// TIA Portal V20 export
DATA_BLOCK "Side_Shifters_SS1"   // DB26
// stored: InstanceOfName Side_Shifters, InstanceOfType FB
"Side_Shifters"
   // VAR_INPUT
   //    set_Hydraulic_Up { ExternalAccessible := 'False'; ExternalVisible := 'False'; ExternalWritable := 'False'} : Bool;
   //    set_Hydraulic_Down { ExternalAccessible := 'False'; ExternalVisible := 'False'; ExternalWritable := 'False'} : Bool;
   //    set_SL_Hydraulic_Up : Bool;
   //    set_SL_Hydraulic_Down : Bool;
   //    set_SR_Hydraulic_Up : Bool;
   //    set_SR_Hydraulic_Down : Bool;
   //    set_SL_Hydraulic_Unit : Bool;
   //    set_SR_Hydraulic_Unit : Bool;
   //    set_Go_To_ST1 : Bool;
   //    set_Go_To_ST2 : Bool;
   //    set_Go_To_ST3 : Bool;
   //    set_Go_To_ST4 : Bool;
   //    ST1_Empty : Bool;
   //    ST2_Empty : Bool;
   //    ST3_Empty : Bool;
   //    ST4_Empty : Bool;
   //    Homing_1_SR : Int;
   //    Homing_2_SR : Int;
   //    Homing_3_SR : Int;
   //    Homing_4_SR : Int;
   //    Homing_1_SL : Int;
   //    Homing_2_SL : Int;
   //    Homing_3_SL : Int;
   //    Homing_4_SL : Int;
   //    SL_Drive_Forward : Bool;
   //    SL_Drive_Backward : Bool;
   //    SR_Drive_Forward : Bool;
   //    SR_Drive_Backward : Bool;
   //    iSL_Sen_Drv_1 : Bool;
   //    iSL_Sen_Drv_2 : Bool;
   //    iSL_Sen_Drv_3 : Bool;
   //    iSL_Sen_Drv_4 : Bool;
   //    iSR_Sen_Drv_1 : Bool;
   //    iSR_Sen_Drv_2 : Bool;
   //    iSR_Sen_Drv_3 : Bool;
   //    iSR_Sen_Drv_4 : Bool;
   //    iSL_Sen_Val1_Up : Bool;
   //    iSL_Sen_Val1_Down : Bool;
   //    iSL_Sen_Val2_Up : Bool;
   //    iSL_Sen_Val2_Down : Bool;
   //    iSR_Sen_Val1_Up : Bool;
   //    iSR_Sen_Val1_Down : Bool;
   //    iSR_Sen_Val2_Up : Bool;
   //    iSR_Sen_Val2_Down : Bool;
   //    iSL_Distance : Int;
   //    iSR_Correct : Int;
   //    iSR_Distance : Int;
   //    iSL_Hydraulic_Filtr : Bool;
   //    iSR_Hydraulic_Empty : Bool;
   //    HWIdentSL : HW_IO;
   //    HWIdentSR : HW_IO;
   //    Reset_Drive : Bool;
   //    Reset_Hydro : Bool;
   // END_VAR
   // VAR_OUTPUT
   //    oSL_Valve_Up { ExternalAccessible := 'False'; ExternalVisible := 'False'; ExternalWritable := 'False'} : Bool;
   //    oSL_Valve_Down { ExternalAccessible := 'False'; ExternalVisible := 'False'; ExternalWritable := 'False'} : Bool;
   //    oSL_Hydraulic_Unit { ExternalAccessible := 'False'; ExternalVisible := 'False'; ExternalWritable := 'False'} : Bool;
   //    oSR_Valve_Up { ExternalAccessible := 'False'; ExternalVisible := 'False'; ExternalWritable := 'False'} : Bool;
   //    oSR_Valve_Down { ExternalAccessible := 'False'; ExternalVisible := 'False'; ExternalWritable := 'False'} : Bool;
   //    oSR_Hydraulic_Unit { ExternalAccessible := 'False'; ExternalVisible := 'False'; ExternalWritable := 'False'} : Bool;
   //    oHydraulic_Status_LED_UP_1 : Bool;
   //    oHydraulic_Status_LED_UP_2 : Bool;
   //    oHydraulic_Status_LED_DOWN_1 : Bool;
   //    oHydraulic_Status_LED_DOWN_2 : Bool;
   //    oSL_Communication_OK : Bool;
   //    oSR_Communication_OK : Bool;
   //    oSL_Forward_Flag : Bool;
   //    oSL_Backward_Flag : Bool;
   //    oSR_Forward_Flag : Bool;
   //    oSR_Backward_Flag : Bool;
   //    oST1_1_Move_Flag : Bool;
   //    oST1_2_Move_Flag : Bool;
   //    oST2_1_Move_Flag : Bool;
   //    oST2_2_Move_Flag : Bool;
   //    oST3_1_Move_flag : Bool;
   //    oST3_2_Move_Flag : Bool;
   //    oST4_1_Move_Flag : Bool;
   //    oST4_2_Move_Flag : Bool;
   // END_VAR
   // VAR_IN_OUT
   //    iSL_Drive_Param : "SEW_MOVIKIT_VelocityDrive_STATUS_V2.1";
   //    iSR_Drive_Param : "SEW_MOVIKIT_VelocityDrive_STATUS_V2.1";
   //    oSL_Drive_Param : "SEW_MOVIKIT_VelocityDrive_SETPOINTS_V2.1";
   //    oSR_Drive_Param : "SEW_MOVIKIT_VelocityDrive_SETPOINTS_V2.1";
   // END_VAR
   // VAR
   //    Hydraulic_SL { ExternalAccessible := 'False'; ExternalVisible := 'False'; ExternalWritable := 'False'} : "Side_Hydraulic";
   //    Hydraulic_SR { ExternalAccessible := 'False'; ExternalVisible := 'False'; ExternalWritable := 'False'} : "Side_Hydraulic";
   //    Side_Driver_Instance { S7_SetPoint := 'True'} : "Side_Driver";
   //    Side_Shifter_Auto_Instance { S7_SetPoint := 'True'} : "Side_Shifter_Auto";
   //    SL_Auto_Speed { S7_SetPoint := 'True'} : Int;
   //    SR_Auto_Speed { S7_SetPoint := 'True'} : Int;
   //    SL_Auto_Forward : Bool;
   //    SL_Auto_Backward : Bool;
   //    SR_Auto_Forward : Bool;
   //    SR_Auto_Backward : Bool;
   //    SR_Distance_Correct : Int;
   //    SL_Error_Laser : Bool;
   //    SR_Error_Laser : Bool;
   //    SL_SR_InPosition : Bool;
   //    SL_Sen_Up : Bool;
   //    SL_Sen_Down : Bool;
   //    SR_Sen_Up : Bool;
   //    SR_Sen_Down : Bool;
   //    SL_Error_Hyd : Bool;
   //    SR_Error_Hyd : Bool;
   //    Error_Drive : Bool;
   //    Error_Hydro : Bool;
   //    Status_Sen_Up : Bool;
   //    Status_Sen_Down : Bool;
   //    RL_Speed : Int;
   //    RR_Speed : Int;
   //    Step_Move_Pallets : Int;
   //    Row_Start : Int;
   //    Row_Destination : Int;
   //    Column_Start : Int;
   //    Column_Destination : Int;
   //    TON_iSR_Error { S7_SetPoint := 'True'} : TON_TIME;
   //    TON_iSL_Error { S7_SetPoint := 'True'} : TON_TIME;
   // END_VAR
BEGIN
END_DATA_BLOCK
